{attribute addProperty BoxType "EL3423-0000-0016"}
{attribute addProperty Id "Active_EnergyAT %I*LINT64818Active_Positive_EnergyAT %I*ULINT64819Active_Negative_EnergyAT %I*ULINT64820"}
{attribute addProperty CRC "270995233"}
{attribute addProperty SizeInBites "192"}
{attribute addProperty SizeInBytes "24"}
TYPE Total_Active_10270F21 :
STRUCT
	{attribute addProperty Name "Active_Energy"}
	Active_Energy AT %I* : LINT;
	{attribute addProperty Name "Active_Positive_Energy"}
	Active_Positive_Energy AT %I* : ULINT;
	{attribute addProperty Name "Active_Negative_Energy"}
	Active_Negative_Energy AT %I* : ULINT;
END_STRUCT
END_TYPE

(* stored: Version 1.2.0.0, ProductVersion 3.1.4024.9
   DUT Total_Active_10270F21: Id {d4796d36-7431-4a84-ad64-7178e0170e35} *)
